(* CODESYS project alimentador.project

Project tree, tasks and I/O mapping:
  Device : CODESYS Control Win V3, 3S - Smart Software Solutions GmbH, order no. 305021, version 3.5.11.30
    application Application
      libraries: Standard, * (System)
      task MainTask (cyclic, interval t#20ms, priority 1) calls PLC_PRG
      task VISU_TASK (cyclic, interval 100 ms, priority 31) calls VisuElems.Visu_Prg
      program PLC_PRG [ST]
      visualisation Visualization
  text list GlobalTextList
*)

// Device/Application/PLC_PRG
PROGRAM PLC_PRG
VAR
	
	ON_OFF: BOOL; //BOTÃO LIGA/DESLIGA
	S1: BOOL; //INDICA SE HA RAÇÃO DENTRO DO COMPARTIMENTO
	//VARIAVEIS AUXILIAR UTILIZADAS 
	AUX_INIT: BOOL;
	AUX2: BOOL;
	
	//TRIGS DO SISTEMA
	R1: R_TRIG;
	Q1: BOOL;
	
	R2: R_TRIG;
	Q2: BOOL;
	
	R3: R_TRIG;
	Q3: BOOL;
	
	R4: R_TRIG;
	Q4: BOOL;
	
	R5: R_TRIG;
	Q5: BOOL;
	
	R6: R_TRIG;
	Q6: BOOL;
	
	R7: R_TRIG;
	Q7: BOOL;
	
	R8: R_TRIG;
	Q8: BOOL;
	
	R9: R_TRIG;
	Q9: BOOL;
	
	R10: R_TRIG;
	Q10: BOOL;
	
	R11: R_TRIG;
	Q11: BOOL;
	
	R12: R_TRIG;
	Q12: BOOL;
	
	R13: R_TRIG;
	Q13: BOOL;
	
	R14: R_TRIG;
	Q14: BOOL;
	
	//TIMES DO SISTEMA
	T1: TOF;
	T1Q: BOOL;
	TIME1: TIME;
	
	T2: TOF;
	T2Q: BOOL;
	TIME2: TIME;
	
	T3: TOF;
	T3Q: BOOL;
	TIME3: TIME;
	
	TWO_HOURS: BOOL;
	FOUR_HOURS: BOOL;
	SIX_HOURS: BOOL;
	EIGHT_HOURS: BOOL;
	TEN_HOURS: BOOL;
	START: BOOL; //INICIA A CONTAGEM
	RELEASE: BOOL;
	
	SET_TIME: TIME; //TEMPO DEFINIDO PELO USUARIO
	L1: BOOL; //SISTEMA LIGADO
	L2: BOOL; //SISTEMA DESLIGADO
	L3: BOOL; //POUCA OU SEM RAÇÃO NO COMPARTIMENDO
	L4: BOOL; //MOTOR RODANDO
	KM1: BOOL;
END_VAR

R1(CLK:=ON_OFF,  Q=>Q1);
R2(CLK:=TWO_HOURS,  Q=>Q2);
R3(CLK:=FOUR_HOURS,  Q=>Q3);
R4(CLK:=SIX_HOURS,  Q=>Q4);
R5(CLK:=EIGHT_HOURS,  Q=>Q5);
R6(CLK:=TEN_HOURS,  Q=>Q6);
R7(CLK:=START OR Q11,  Q=>Q7);
R8(CLK:=AUX2,  Q=>Q8);
R9(CLK:=NOT(T1Q),  Q=>Q9);
R10(CLK:=Q9,  Q=>Q10);
R11(CLK:=NOT(T2Q),  Q=>Q11);
R12(CLK:=RELEASE,  Q=>Q12);
R13(CLK:=NOT T3Q,  Q=>Q13);
R14(CLK:=NOT(AUX_INIT),  Q=>Q14);

IF Q1 THEN
	AUX_INIT := NOT(AUX_INIT);
END_IF

IF AUX_INIT THEN 
	L1:=TRUE;
	L2:=FALSE;
	IF Q2 THEN
		SET_TIME:= T#2H;
	END_IF
	
	IF Q3 THEN
		SET_TIME:= T#4H;
	END_IF
	
	IF Q4 THEN
		SET_TIME:= T#6H;
	END_IF
	
	IF Q5 THEN
		SET_TIME:= T#8H;
	END_IF
	
	IF Q6 THEN
		SET_TIME:= T#10H;
	END_IF
	
	IF Q7 AND (SET_TIME>T#0H) THEN 
		AUX2:=TRUE;
	END_IF
	
	IF Q9 THEN
		KM1:=TRUE;
		L4:= TRUE;
	END_IF
	
	IF Q11 THEN
		KM1:=FALSE;
		AUX2:=FALSE;
		L4:= FALSE;
	END_IF
	
	IF Q12 THEN
		KM1:=TRUE;
		L4:= TRUE;
	END_IF
	
	IF Q13 THEN
		KM1:=FALSE;
		L4:= FALSE;
	END_IF
	IF (NOT S1) THEN
		L1:=FALSE;
		L2:=FALSE;
		L3:=TRUE;
		ELSE
			L3:=FALSE;
	END_IF
	ELSE
		L1:=FALSE;
		L2:=TRUE;
		L3:=FALSE;
END_IF

T1(IN:=Q8, PT:=SET_TIME, Q=>T1Q,ET=>TIME1);
T2(IN:=Q10, PT:=T#5S, Q=>T2Q,ET=>TIME2);
T3(IN:=Q12, PT:=T#5S, Q=>T3Q,ET=>TIME3);

END_PROGRAM

// Device/Application/Visualization
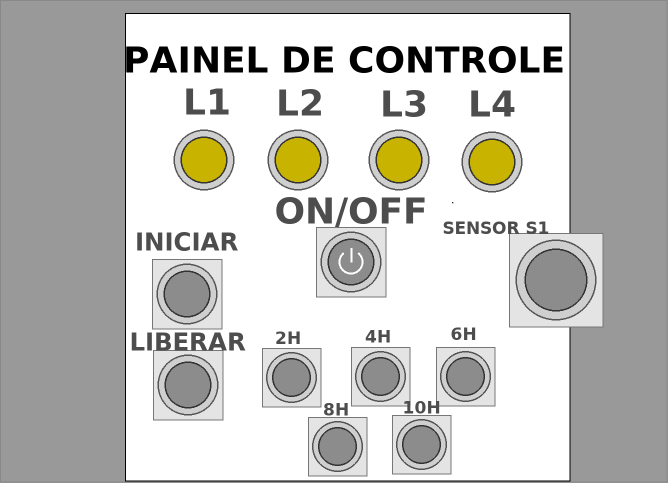
VISUALIZATION Visualization  // 668x483
    RoundedRectangle (125,13 445x468)
    Lamp1 (169,125 70x70), variable: PLC_PRG.L1, style: Lamp-Lamp1-Yellow
    Lamp1 (263,125 70x70), variable: PLC_PRG.L2, style: Lamp-Lamp1-Yellow
    Lamp1 (364,125 70x70), variable: PLC_PRG.L3, style: Lamp-Lamp1-Yellow
    PushSwitch (153,350 70x70), variable: PLC_PRG.RELEASE, behaviour: TOGGLE, style: Switch-PushSwitch-Gray
    PowerSwitch (316,227 70x70), variable: PLC_PRG.ON_OFF, behaviour: TOGGLE, style: Switch-PowerSwitch-Gray
    PushSwitch (152,259 70x70), variable: PLC_PRG.START, behaviour: TOGGLE, style: Switch-PushSwitch-Gray
    Lamp1 (457,127 70x70), variable: PLC_PRG.L4, style: Lamp-Lamp1-Yellow
    Label (426,234 150x30)
    Label (183,72 48x60), "L1"
    Label (283,105 34x30)
    Label (322,105 150x30)
    PushSwitch (452,202 1x1), behaviour: TOGGLE, style: Switch-PushSwitch-Gray
    PushSwitch (446,233 220x94), variable: PLC_PRG.S1, behaviour: TOGGLE, style: Switch-PushSwitch-Gray
    PushSwitch (261,348 61x59), variable: PLC_PRG.TWO_HOURS, behaviour: TOGGLE, style: Switch-PushSwitch-Gray
    PushSwitch (350,347 61x59), variable: PLC_PRG.FOUR_HOURS, behaviour: TOGGLE, style: Switch-PushSwitch-Gray
    PushSwitch (435,347 61x59), variable: PLC_PRG.SIX_HOURS, behaviour: TOGGLE, style: Switch-PushSwitch-Gray
    PushSwitch (307,417 61x59), variable: PLC_PRG.EIGHT_HOURS, behaviour: TOGGLE, style: Switch-PushSwitch-Gray
    PushSwitch (391,415 61x59), variable: PLC_PRG.TEN_HOURS, behaviour: TOGGLE, style: Switch-PushSwitch-Gray
    Label (359,74 90x60), "L3"
    Label (255,73 90x60), "L2"
    Label (447,74 90x60), "L4"
    Label (259,181 184x60), "ON/OFF"
    Label (77,312 222x60), "LIBERAR"
    Label (76,212 222x60), "INICIAR"
    Label (385,198 222x60), "SENSOR S1"
    Label (270,308 36x60), "2H"
    Label (364,311 28x51), "4H"
    Label (443,304 41x60), "6H"
    Label (322,384 28x51), "8H"
    Label (396,382 51x51), "10H"
    Label (44,30 600x60), "PAINEL DE CONTROLE"
END_VISUALIZATION
